SYSTEM Test Big Computation ser 40
  (* Version 1.0, 2005-12-23, Goran Cengic, Chalmers *)
  DEVICE Test Device : DeviceType_not_used
    RESOURCE Test Resource : ResourceType_not_used
      FBS
        restart : E_RESTART;
        stop : E_STOP;
        big1 : BigComputation;
        big2 : BigComputation;
        big3 : BigComputation;
        big4 : BigComputation;
        big5 : BigComputation;
        big6 : BigComputation;
        big7 : BigComputation;
        big8 : BigComputation;
        big9 : BigComputation;
        big10 : BigComputation;
        big11 : BigComputation;
        big12 : BigComputation;
        big13 : BigComputation;
        big14 : BigComputation;
        big15 : BigComputation;
        big16 : BigComputation;
        big17 : BigComputation;
        big18 : BigComputation;
        big19 : BigComputation;
        big20 : BigComputation;
        big21 : BigComputation;
        big22 : BigComputation;
        big23 : BigComputation;
        big24 : BigComputation;
        big25 : BigComputation;
        big26 : BigComputation;
        big27 : BigComputation;
        big28 : BigComputation;
        big29 : BigComputation;
        big30 : BigComputation;
        big31 : BigComputation;
        big32 : BigComputation;
        big33 : BigComputation;
        big34 : BigComputation;
        big35 : BigComputation;
        big36 : BigComputation;
        big37 : BigComputation;
        big38 : BigComputation;
        big39 : BigComputation;
        big40 : BigComputation;
      END_FBS
      EVENT_CONNECTIONS
        restart.COLD TO big1.EI;
        big1.EO TO big2.EI;
        big2.EO TO big3.EI;
        big3.EO TO big4.EI;
        big4.EO TO big5.EI;
        big5.EO TO big6.EI;
        big6.EO TO big7.EI;
        big7.EO TO big8.EI;
        big8.EO TO big9.EI;
        big9.EO TO big10.EI;
        big10.EO TO big11.EI;
        big11.EO TO big12.EI;
        big12.EO TO big13.EI;
        big13.EO TO big14.EI;
        big14.EO TO big15.EI;
        big15.EO TO big16.EI;
        big16.EO TO big17.EI;
        big17.EO TO big18.EI;
        big18.EO TO big19.EI;
        big19.EO TO big20.EI;
        big20.EO TO big21.EI;
        big21.EO TO big22.EI;
        big22.EO TO big23.EI;
        big23.EO TO big24.EI;
        big24.EO TO big25.EI;
        big25.EO TO big26.EI;
        big26.EO TO big27.EI;
        big27.EO TO big28.EI;
        big28.EO TO big29.EI;
        big29.EO TO big30.EI;
        big30.EO TO big31.EI;
        big31.EO TO big32.EI;
        big32.EO TO big33.EI;
        big33.EO TO big34.EI;
        big34.EO TO big35.EI;
        big35.EO TO big36.EI;
        big36.EO TO big37.EI;
        big37.EO TO big38.EI;
        big38.EO TO big39.EI;
        big39.EO TO big40.EI;
        big40.EO TO stop.STOP;
      END_CONNECTIONS
    END_RESOURCE
  END_DEVICE
END_SYSTEM
